// TIA Portal V19 export
TYPE "C701_VAR_IF_KLB_TYPIC"
   STRUCT
      KLB_TOE { ExternalAccessible := 'False'; ExternalVisible := 'False'; ExternalWritable := 'False'} : Bool;   // Brandklep gesloten
   END_STRUCT;
END_TYPE
